//Status information specific to the cabinet IPC --> PNOZ, can be customized depending on cabinet
TYPE ST_MCC_CustomStatusOut :
STRUCT
    bit16_Reserved: BIT;
    bit17_Reserved: BIT;
    bit18_Reserved: BIT;
    bit19_Reserved: BIT;
    bit20_FocusDoorLocked: BIT;
    bit21_Reserved: BIT;
    bit22_ChangerMovingPos: BIT; //Set if moving in a positive direction
    bit23_ChangerMovingNeg: BIT; //Set if moving in a negative direction
    bit24_Reserved: BIT;
    bit25_Reserved: BIT;
    bit26_Reserved: BIT;
    bit27_Reserved: BIT;
    bit28_Reserved: BIT;
    bit29_Reserved: BIT;
    bit30_Reserved: BIT;
    bit31_Reserved: BIT;
END_STRUCT
END_TYPE

(* stored: Version 1.1.0.1
   DUT ST_MCC_CustomStatusOut: Id {6d8ad02a-be6f-0232-209b-380247c69933} *)
